// TIA Portal V18 export
TYPE "OP40_Data"
   STRUCT
      AssemblyResult : Byte;
      SN : String[30];
      ProcessData { S7_SetPoint := 'True'} : "WriteProcessData";
   END_STRUCT;
END_TYPE
